Fanuc KAREL source: kt00858.compact.KL

PROGRAM KT00858
%STACKSIZE=65535
%PRIORITY=65535
%NOLOCKGROUP
VAR
R1 : REAL
R2 : REAL
OUT : INTEGER
BEGIN
R1=2.0
R2=3.0
R1=2.0
R2=3.0
OUT=ROUND(R1)
END KT00858
